PROGRAM prgEMS
VAR PERSISTENT
	byMaxDepthOfDischrgEPO		: BYTE;							//{#lynus.ag#()}
	byPrioMinChrgBattSOCInEPO	: BYTE;							//{#lynus.ag#()}
	byResChrgfromGridToBatt		: BYTE;							//{#lynus.ag#()}
	byResChrgfromGridToBatt_Controlled		: BYTE;							//{#lynus.ag#()}
	byReserveSOCEPO				: BYTE;							//{#lynus.ag#()}
	uiUpdateTime				: UINT;							//{#lynus.ag#()}
	bEnableEMS					: BOOL;							//{#lynus.ag#()}
	bAllowChrgFromGrid			: BOOL;							//{#lynus.ag#()}
	rMainFuseCSEMS				: REAL;							//{#lynus.ag#()}
	iOperationModeEMS			: INT;							//{#lynus.ag#()}
END_VAR
VAR
	fbEMS						: FB_EMS_T;
	bIsEnableEMS				: BOOL;							//{#lynus.ag#()}
	bStateAllowChrgFromGrid		: BOOL;							//{#lynus.ag#()}
	bHPActivate					: BOOL;							//{#lynus.ag#()}
	bControllingState			: BOOL;							//{#lynus.ag#()}
	iMessageEMS					: INT;							//{#lynus.ag#()}
	rHeartbeatEMS				: REAL;							//{#lynus.ag#()}
	rErrorWarningEMS			: REAL;							//{#lynus.ag#()}
	rReadyEMS					: REAL;							//{#lynus.ag#()}
	rNewBatteryPowerEMS			: REAL;							//{#lynus.ag#()}
	b_EnableBatteryChargingControl				: BOOL:=TRUE;																						//{#lynus.ag#()} //  
	b_StartReleaseBatteryCharging				: BOOL;																								//{#lynus.ag#()} //  
	b_StopReleaseBatteryCharging				: BOOL;																								//{#lynus.ag#()} //  
	b_TimeBasedReleaseChargingBattery			: BOOL;																								//{#lynus.ag#()} //  
	b_StartChargingfor3Hours					: BOOL;																								//{#lynus.ag#()} //  

	RS_ChargingFromGridAllowed: Rs;
	tof_3HourCharging: Tof;
	RS_3HourCharging: Rs;
	r_trig_3HourChraging: R_trig;
	f_trig_3HourChragingOver: f_trig;
	m_PIDBatterySC_Enabled: BOOL;
	m_PIDBatteryPLCLM_Dischrg_Enabled: BOOL;
	m_fbPIDBatteryPLCLM_Chrg_Enabled: BOOL;
	m_fbPIDBatteryEPO_Enabled: BOOL;
END_VAR

// Stefan 21.02.2024
// disabled bControllingState to make sure the backend is not regulating the battery
// changeed lacal EMS PID regulator for charging and discharging in FB_EMS_T to fullfill the PTM requirements to fixie PID parameters, made the regulator slower for more stability. 

fbEMS.stSetupEMS.bAllowChrgFromGrid := bAllowChrgFromGrid;
fbEMS.stSetupEMS.byMaxDepthOfDischrgEPO := byMaxDepthOfDischrgEPO;
fbEMS.stSetupEMS.byPrioMinChrgBattSOCInEPO := byPrioMinChrgBattSOCInEPO;
fbEMS.stSetupEMS.byReserveSOCEPO := byReserveSOCEPO;
fbEMS.stSetupEMS.rSizeMainFuseCS := rMainFuseCSEMS;
fbEMS.stSetupEMS.uiUpdateTime := uiUpdateTime;

IF iOperationModeEMS = 0 THEN fbEMS.eOperationMode := E_OperatingMode_EMS.eAllOff;
ELSIF iOperationModeEMS = 1 THEN fbEMS.eOperationMode := E_OperatingMode_EMS.eSelfConsumption;	
ELSIF iOperationModeEMS = 2 THEN fbEMS.eOperationMode := E_OperatingMode_EMS.ePeakLoadCapping;
ELSIF iOperationModeEMS = 3 THEN fbEMS.eOperationMode := E_OperatingMode_EMS.eLoadManagement;			
END_IF

fbEMS(
	bEnable						:= bEnableEMS, 
	diNrOfEM_IN_ECS				:= , 
	stSetupEMS					:= , 
	eOperationMode				:= , 
	eSpeedModeBackendController	:= E_SpeedModeBackendController_EMS.eFast, 
	eSpeedModeLocalController	:= E_SpeedModeLocalController_EMS.eFast,
	bActivateHP					:= bHPActivate, 
	bControllingState			:= TRUE, //bControllingState, 
	rHeartbeat					:= rHeartbeatEMS, 
	rErrorWarning				:= rErrorWarningEMS, 
	rEnergyOptReady				:= rReadyEMS, 
	rNewBattPower				:= rNewBatteryPowerEMS, 
	b_ZeroPowerRegulation		:=,
	b_EnableBatteryChargingControl	:= TRUE,
	b_StartReleaseBatteryCharging 	:= TRUE,
	b_StopReleaseBatteryCharging 	:= ,
	rMaxBattChargingPower			:= SEL(bAllowChrgFromGrid,100,63),	// 80 kW = 100%, 63 % = 50 kW
	rPeakDetectionforCalculation 	:= 20,	// was original 3, caused issues that load management not caluculeted. see EMS line 313
	
	eMessageEMS				=> iMessageEMS, 
	bStateEnable			=> bIsEnableEMS, 
	bStateAllowChrgFromGrid	=> bStateAllowChrgFromGrid, 
	bMissingPowerData		=> , 
	bSurplusAvailable		=> , 
	byProgress				=> , 
	uiState_OUT				=> , 
	diNrOfEMS_OUT			=> , 
	arrMinPrioReached		=> , 
	arrMaxPrioReached		=> ,
	b_TimeBasedReleaseChargingBattery => b_TimeBasedReleaseChargingBattery);
	
	// update 20230228 
	// charging control done with bAllowChrgFromGrid: Charging is allways allowed (If surplus is available) , but charging from grid is only allowed during the night time. 
// b_EnableBatteryChargingControl
// b_StartReleaseBatteryCharging
// b_StopReleaseBatteryCharging
// fbEMS.stSetupEMS.bAllowChrgFromGrid := bAllowChrgFromGrid;
RS_ChargingFromGridAllowed( SET := b_EnableBatteryChargingControl AND b_StartReleaseBatteryCharging,
							Reset1 := NOT b_EnableBatteryChargingControl OR (b_EnableBatteryChargingControl AND b_StopReleaseBatteryCharging));

r_trig_3HourChraging( 	clk:=b_StartChargingfor3Hours);
f_trig_3HourChragingOver( clk:=tof_3HourCharging.Q);

tof_3HourCharging(	IN:= r_trig_3HourChraging.Q,
					PT := T#3H);
RS_3HourCharging(	Set := r_trig_3HourChraging.Q,
					Reset1 := f_trig_3HourChragingOver.Q OR (r_trig_3HourChraging.Q AND RS_3HourCharging.Q1) OR prgBattery.dwSOCBattery > byResChrgfromGridToBatt_Controlled);
							
							
IF b_EnableBatteryChargingControl AND (RS_ChargingFromGridAllowed.Q1 OR RS_3HourCharging.Q1) THEN
	bAllowChrgFromGrid := TRUE;
	fbEMS.stSetupEMS.byResChrgfromGridToBatt := byResChrgfromGridToBatt_Controlled; // battery max soc according input field when charging the battery in the night
ELSE
	bAllowChrgFromGrid := FALSE;
	fbEMS.stSetupEMS.byResChrgfromGridToBatt := byResChrgfromGridToBatt;			// battery max SOC according to EMS setting, e.g. 100%; this should only get achieved by grid surplus
END_IF
 
// find out which regulator is active

m_PIDBatterySC_Enabled := fbEMS.fbPIDBatterySC.bEnable;;
m_PIDBatteryPLCLM_Dischrg_Enabled := fbEMS.fbPIDBatteryPLCLM_Dischrg.bEnable;
m_fbPIDBatteryPLCLM_Chrg_Enabled := fbEMS.fbPIDBatteryPLCLM_Chrg.bEnable;
m_fbPIDBatteryEPO_Enabled := fbEMS.fbPIDBatteryEPO.bEnable;

END_PROGRAM

(* stored: Version 1.1.0.1, ProductVersion 3.1.4024.12
   POU prgEMS: Id {6f701af2-5d23-45b1-901b-ca5d2d305ed9}, SpecialFunc None *)
